// TIA Portal V20 export
DATA_BLOCK "ET500SP_502"   // DB231
// stored: MemoryReserve 100
   VAR
      SPARE1 : Bool;
      SPARE2 : Bool;
      SPARE3 : Bool;
      SPARE4 : Bool;
      SPARE5 : Bool;
      SPARE6 : Bool;
      SPARE7 : Bool;
      SPARE8 : Bool;
      SPARE9 : Bool;
      SPARE10 : Bool;
      SPARE11 : Bool;
      SPARE12 : Bool;
      SPARE13 : Bool;
      SPARE14 : Bool;
      SPARE15 : Bool;
      SPARE16 : Bool;
   END_VAR
BEGIN
END_DATA_BLOCK
